INTERFACE ITF_BaseControlElementDecoratorParent EXTENDS ITF_BaseControlElement

END_INTERFACE

(* stored: Version 1.1.0.1
   Itf ITF_BaseControlElementDecoratorParent: Id {916549e7-ccae-0db7-1dc6-fc3dd7272f1a} *)
